FUNCTION_BLOCK FB_Toggle
VAR_INPUT
END_VAR
VAR_OUTPUT
END_VAR
VAR
	Timer_1s 	: TON; 		// Timer für den Takt
	Timer_500ms	: TON;		// Timer für Ampelblinktakt
	Cycle_1s	: BOOL;		// Tooglevariable
END_VAR

// Timmer 1s Zyklus
Timer_1s(IN:=NOT Timer_1s.Q ,
		 PT:=T#1S );
		 
Cycle_1s := Cycle_1s XOR Timer_1s.Q;

//Timer für Ampelblinktakt
Timer_500ms(IN:=NOT Timer_500ms.Q ,
		 	PT:=T#600MS );
			
bBlink := bBlink XOR Timer_500ms.Q;

END_FUNCTION_BLOCK

(* stored: Version 1.1.0.1, ProductVersion 3.1.4024.12
   POU FB_Toggle: Id {bc35b369-10af-48ab-a6d8-07058ca157a8}, SpecialFunc None *)
